// TIA Portal V19 export
FUNCTION_BLOCK "Sample_alarmed_FB"   // FB1, LAD
TITLE = Alarms -Timed Alarm System
{ S7_Optimized_Access := 'TRUE' }
// stored: MemoryReserve 100, SetENOAutomatically false
   VAR_INPUT
      Alarm_Trigger : Bool;   // Used to Trigger the Alarm Watching
      Timer_PT : Time;   // Time Until Alarm goes off after Trigger
      ACK_Button : Bool;   // Acknowledged Alarm Button
      Reset_Button : Bool;   // Reset Alarm Button
   END_VAR
   VAR_OUTPUT
      Alarm : Bool;   // Current Status of Alarm
      Alarm_ACKED : Bool;   // Alarm Acknowledged (Y/N)
      Alarm_Indicator : Bool;   // Alarm LED Indicator
   END_VAR
   VAR
      Alarm_Timer { S7_SetPoint := 'True'} : TON_TIME;   // Used when Triggering Alarm Active
      Alarm_Timer_Done : Bool;   // Triggers when Alarm Timer Elapsed
      Alarm_Active : Bool;   // Alarm is Active
      Alarm_ACK : Bool;   // Alarm is Acknowledged
      Alarm_Reset : Bool;   // Alarm is Reset
   END_VAR
BEGIN

REGION Network 1: Start Alarm
   // When Alarm_Trigger > Timer_PT the Alarm_Timer is Done
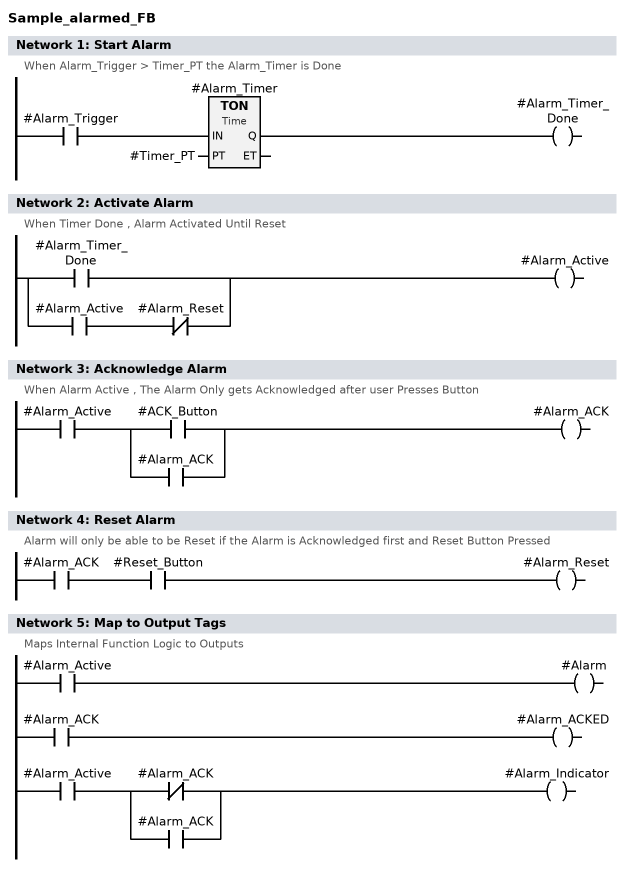
   RUNG wire#powerrail
      Contact( #Alarm_Trigger )
      { S7_Templates := "time_type := Time" } #Alarm_Timer.TON(pt := #Timer_PT, et =>)
      Coil( #Alarm_Timer_Done )
   END_RUNG
   // the same network as SCL:
   #Alarm_Timer(IN := #Alarm_Trigger, PT := #Timer_PT);   // TON
   #Alarm_Timer_Done := #Alarm_Timer.Q;
END_REGION

REGION Network 2: Activate Alarm
   // When Timer Done , Alarm Activated Until Reset
   RUNG wire#powerrail
      Contact( #Alarm_Timer_Done )
      wire#w1
      Coil( #Alarm_Active )
   END_RUNG
   RUNG wire#powerrail
      Contact( #Alarm_Active )
      I_Contact( #Alarm_Reset )
   END_RUNG wire#w1
   // the same network as SCL:
   #Alarm_Active := #Alarm_Timer_Done OR (#Alarm_Active AND NOT #Alarm_Reset);
END_REGION

REGION Network 3: Acknowledge Alarm
   // When Alarm Active , The Alarm Only gets Acknowledged after user Presses Button
   RUNG wire#powerrail
      Contact( #Alarm_Active )
      wire#w1
      Contact( #ACK_Button )
      wire#w2
      Coil( #Alarm_ACK )
   END_RUNG
   RUNG wire#w1
      Contact( #Alarm_ACK )
   END_RUNG wire#w2
   // the same network as SCL:
   #Alarm_ACK := #Alarm_Active AND (#ACK_Button OR #Alarm_ACK);
END_REGION

REGION Network 4: Reset Alarm
   // Alarm will only be able to be Reset if the Alarm is Acknowledged first and Reset Button Pressed
   RUNG wire#powerrail
      Contact( #Alarm_ACK )
      Contact( #Reset_Button )
      Coil( #Alarm_Reset )
   END_RUNG
   // the same network as SCL:
   #Alarm_Reset := #Alarm_ACK AND #Reset_Button;
END_REGION

REGION Network 5: Map to Output Tags
   // Maps Internal Function Logic to Outputs
   RUNG wire#powerrail
      Contact( #Alarm_Active )
      Coil( #Alarm )
   END_RUNG
   RUNG wire#powerrail
      Contact( #Alarm_ACK )
      Coil( #Alarm_ACKED )
   END_RUNG
   RUNG wire#powerrail
      Contact( #Alarm_Active )
      wire#w1
      I_Contact( #Alarm_ACK )
      wire#w2
      Coil( #Alarm_Indicator )
   END_RUNG
   RUNG wire#w1
      Contact( #Alarm_ACK )
   END_RUNG wire#w2
   // the same network as SCL:
   #Alarm := #Alarm_Active;
   #Alarm_ACKED := #Alarm_ACK;
   #Alarm_Indicator := #Alarm_Active AND (NOT #Alarm_ACK OR #Alarm_ACK);
END_REGION

REGION Network 6: Spare
END_REGION
END_FUNCTION_BLOCK
